// TIA Portal V18 export
FUNCTION_BLOCK "Block_801"   // FB11, LAD
{ S7_Optimized_Access := 'TRUE' }
VERSION : 0.1
// stored: AutoNumber true, IsIECCheckEnabled false, IsRetainMemResEnabled false, MemoryReserve 100, SetENOAutomatically false, UDAEnableTagReadback false
BEGIN
END_FUNCTION_BLOCK
